(* PLC project  *)

PROGRAM P

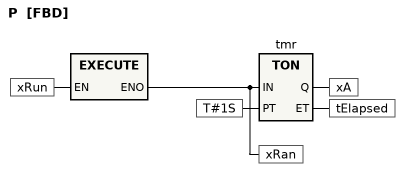
(* FBD diagram, written out as Structured Text *)
IF xRun THEN
  nCount := nCount + 1;
END_IF;
tmr(IN := xRun, PT := T#1S);
xA := tmr.Q;
tElapsed := tmr.ET;
xRan := xRun;
END_PROGRAM
